{attribute addProperty BoxType "EJ3108-0000-0017"}
{attribute addProperty Id "AI_Standard_ChannelAT %I*ARRAY[0..7] OF AI_Standard_Channel_F16A160D256320WcStateAT %I*WcState_F855686C1620InfoDataAT %I*InfoData_BC63D37F80100"}
{attribute addProperty CRC "515865240"}
{attribute addProperty SizeInBites "352"}
{attribute addProperty SizeInBytes "44"}
TYPE EJ3108_86604016 :
STRUCT
	{attribute addProperty Name "AI_Standard_Channel"}
	AI_Standard_Channel : ARRAY[0..7] OF AI_Standard_Channel_F16A160D;
	{attribute addProperty Name "WcState"}
	WcState : WcState_F855686C;
	{attribute addProperty Name "InfoData"}
	InfoData : InfoData_BC63D37F;
END_STRUCT
END_TYPE

(* stored: Version 1.2.0.0, ProductVersion 3.1.4024.9
   DUT EJ3108_86604016: Id {e3ccb3d2-c596-4c3f-adb6-3fb9e8378851} *)
